# EPICS StreamDevice protocol: arduinoepics/abacus_light/device_config/abacus_light.proto
Terminator = CR LF;
replytimeout = 1000;
@mismatch{ in "Invalid command, type help";}

debug{
    out "%s";
    in "%39c";
}

channel_set_read{
    out "ch \$1 ?";
    in "current set state: ch \$1 %{0|1}";
}

channel_set{
    out "ch \$1 %{off|on}";
}

all_channel_off{
    out "all ch %{off}";
}

dimm_read{
    out "dimm \$1 ?";
    in "current dimmer state: ch \$1 %d";
}

dimm_set{
    out "dimm \$1 %d";
}
